{attribute 'qualified_only'}
VAR_GLOBAL
	rAIInput1 : REAL;
	rAIInput2 : REAL;
	
	fSetpointValueToScope : LREAL;
	fActualValueToScope : LREAL;
	foutToScope : LREAL;
	
	outputDischargeValve : REAL;
	scaledDisturbancePotmeter : REAL;
	
	StartStep5 : BOOL;
	StartStep10 : BOOL;
	StartStep15 : BOOL;
	
	setManual : BOOL;
	setAuto : BOOL;
	
END_VAR

(* stored: Version 1.1.0.1, ProductVersion 3.1.4024.13
   GVL GVL: Id {ef375329-646c-4fe3-ba82-2432ee535fa0} *)
